PROGRAM TemperatureSensorEx2
VAR
	fbHVACTemperatureSensorEx2: FB_HVACTemperatureSensorEx2;
	eDataSecurityType: E_HVACDataSecurityType;
	bSetDefault: BOOL;
	bEnable: BOOL;
	iRawValue: INT;
	byStatusRawValue: BYTE;
	iConversionFactor: INT;
	bEnableLimitCtrl: BOOL;
	bReset: BOOL;
	rOffset: REAL;
	rHighLimit: REAL;
	rLowLimit: REAL;
	rReplacementValue: REAL;
	rSmoothFactor: REAL;
	iTemperatureSensorMode: INT;
	rPresentValue: REAL;
	bErrorGeneral: BOOL;
	udiError: UDINT;
	bErrorSensor: BOOL;
	bErrorHighLimit: BOOL;
	bErrorLowLimit: BOOL;
	bErrorConversionFactor: BOOL;
	bInvalidParameter: BOOL;
END_VAR

fbHVACTemperatureSensorEx2(
	eDataSecurityType:=eDataSecurityType, 
	bSetDefault:=bSetDefault, 
	bEnable:=bEnable, 
	iRawValue:=iRawValue, 
	byStatusRawValue:=byStatusRawValue, 
	iConversionFactor:=iConversionFactor, 
	bEnableLimitCtrl:=bEnableLimitCtrl, 
	bReset:=bReset, 
	rPresentValue=>rPresentValue, 
	bErrorGeneral=>bErrorGeneral, 
	udiError=>udiError, 
	bErrorSensor=>bErrorSensor, 
	bErrorHighLimit=>bErrorHighLimit, 
	bErrorLowLimit=>bErrorLowLimit, 
	bErrorConversionFactor=>bErrorConversionFactor, 
	bInvalidParameter=>bInvalidParameter, 
	rOffset:=rOffset, 
	rHighLimit:=rHighLimit, 
	rLowLimit:=rLowLimit, 
	rReplacementValue:=rReplacementValue, 
	rSmoothFactor:=rSmoothFactor, 
	iTemperatureSensorMode:=iTemperatureSensorMode);

END_PROGRAM

(* stored: Version 1.1.0.1, ProductVersion 3.1.4024.3
   POU TemperatureSensorEx2: Id {b03110b6-15c7-4a96-83f5-3e5144d93627}, SpecialFunc None *)
